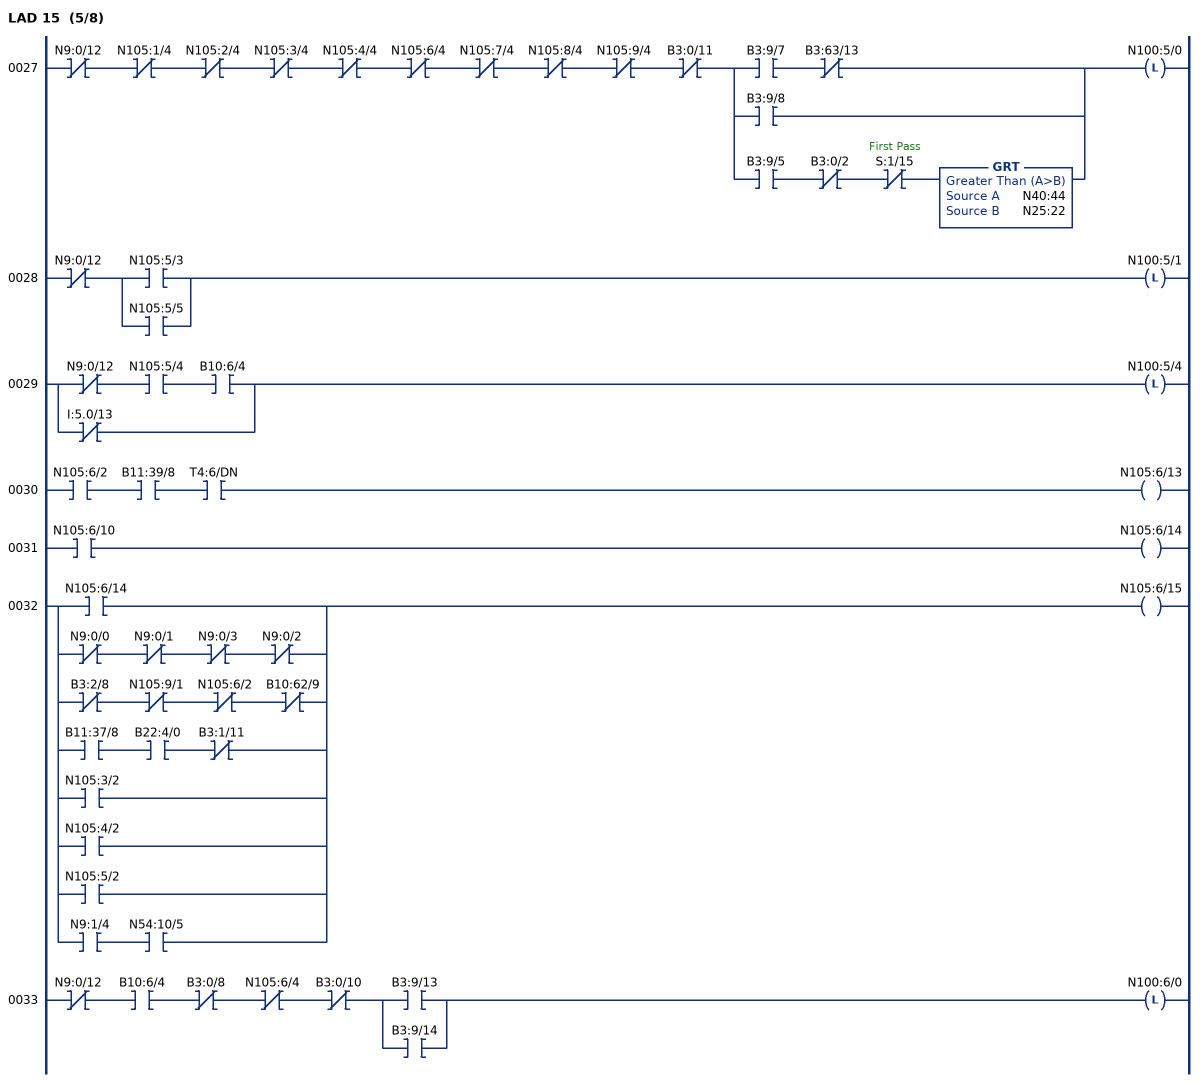
% Rung: 27 %
SOR XIO N9:0/12 XIO N105:1/4 XIO N105:2/4 XIO N105:3/4 XIO N105:4/4 XIO N105:6/4 XIO N105:7/4 XIO N105:8/4 XIO N105:9/4 XIO B3:0/11 BST XIC B3:9/7 XIO B3:63/13 NXB XIC B3:9/8 NXB XIC B3:9/5 XIO B3:0/2 XIO S:1/15 GRT N40:44 N25:22 BND OTL N100:5/0 EOR
%   S:1/15  "First Pass" %
% Rung: 28 %
SOR XIO N9:0/12 BST XIC N105:5/3 NXB XIC N105:5/5 BND OTL N100:5/1 EOR
% Rung: 29 %
SOR BST XIO N9:0/12 XIC N105:5/4 XIC B10:6/4 NXB XIO I:5.0/13 BND OTL N100:5/4 EOR
% Rung: 30 %
SOR XIC N105:6/2 XIC B11:39/8 XIC T4:6/DN OTE N105:6/13 EOR
% Rung: 31 %
SOR XIC N105:6/10 OTE N105:6/14 EOR
% Rung: 32 %
SOR BST XIC N105:6/14 NXB XIO N9:0/0 XIO N9:0/1 XIO N9:0/3 XIO N9:0/2 NXB XIO B3:2/8 XIO N105:9/1 XIO N105:6/2 XIO B10:62/9 NXB XIC B11:37/8 XIC B22:4/0 XIO B3:1/11 NXB XIC N105:3/2 NXB XIC N105:4/2 NXB XIC N105:5/2 NXB XIC N9:1/4 XIC N54:10/5 BND OTE N105:6/15 EOR
% Rung: 33 %
SOR XIO N9:0/12 XIC B10:6/4 XIO B3:0/8 XIO N105:6/4 XIO B3:0/10 BST XIC B3:9/13 NXB XIC B3:9/14 BND OTL N100:6/0 EOR

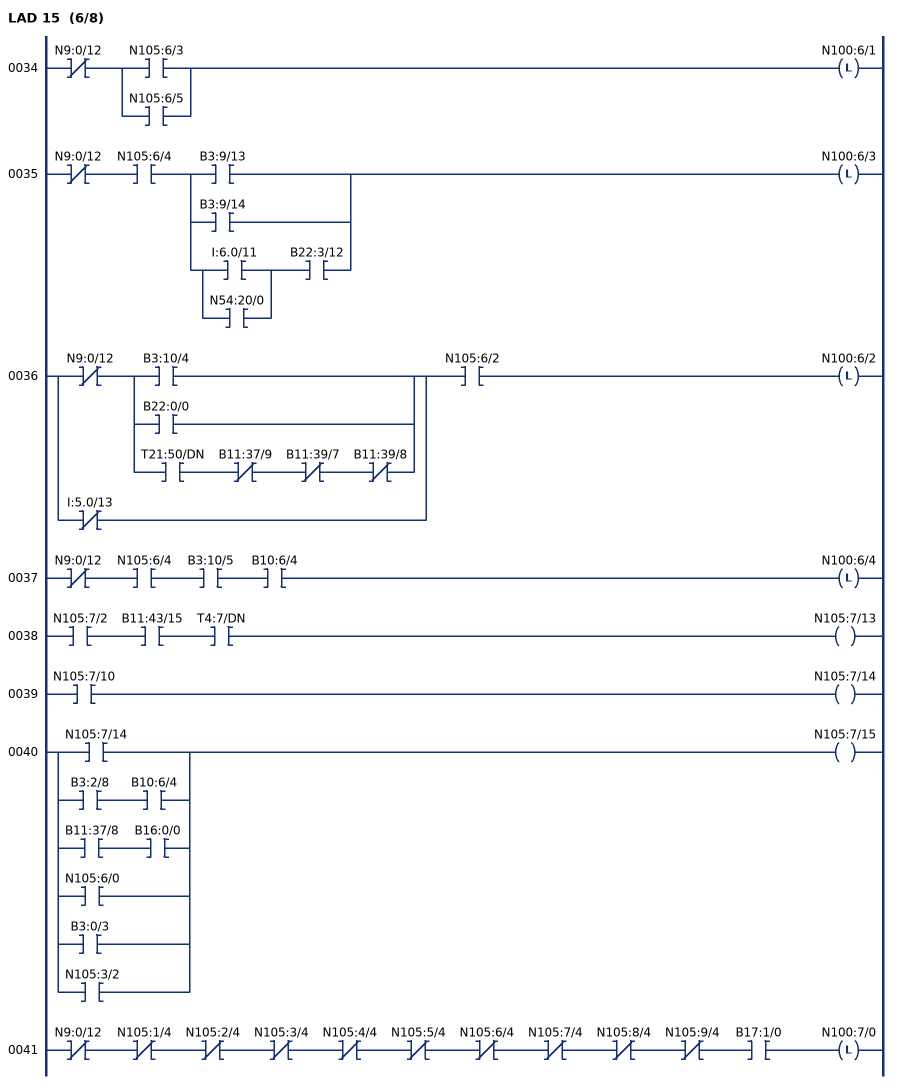
% Rung: 34 %
SOR XIO N9:0/12 BST XIC N105:6/3 NXB XIC N105:6/5 BND OTL N100:6/1 EOR
% Rung: 35 %
SOR XIO N9:0/12 XIC N105:6/4 BST XIC B3:9/13 NXB XIC B3:9/14 NXB BST XIC I:6.0/11 NXB XIC N54:20/0 BND XIC B22:3/12 BND OTL N100:6/3 EOR
% Rung: 36 %
SOR BST XIO N9:0/12 BST XIC B3:10/4 NXB XIC B22:0/0 NXB XIC T21:50/DN XIO B11:37/9 XIO B11:39/7 XIO B11:39/8 BND NXB XIO I:5.0/13 BND XIC N105:6/2 OTL N100:6/2 EOR
% Rung: 37 %
SOR XIO N9:0/12 XIC N105:6/4 XIC B3:10/5 XIC B10:6/4 OTL N100:6/4 EOR
% Rung: 38 %
SOR XIC N105:7/2 XIC B11:43/15 XIC T4:7/DN OTE N105:7/13 EOR
% Rung: 39 %
SOR XIC N105:7/10 OTE N105:7/14 EOR
% Rung: 40 %
SOR BST XIC N105:7/14 NXB XIC B3:2/8 XIC B10:6/4 NXB XIC B11:37/8 XIC B16:0/0 NXB XIC N105:6/0 NXB XIC B3:0/3 NXB XIC N105:3/2 BND OTE N105:7/15 EOR
% Rung: 41 %
SOR XIO N9:0/12 XIO N105:1/4 XIO N105:2/4 XIO N105:3/4 XIO N105:4/4 XIO N105:5/4 XIO N105:6/4 XIO N105:7/4 XIO N105:8/4 XIO N105:9/4 XIC B17:1/0 OTL N100:7/0 EOR

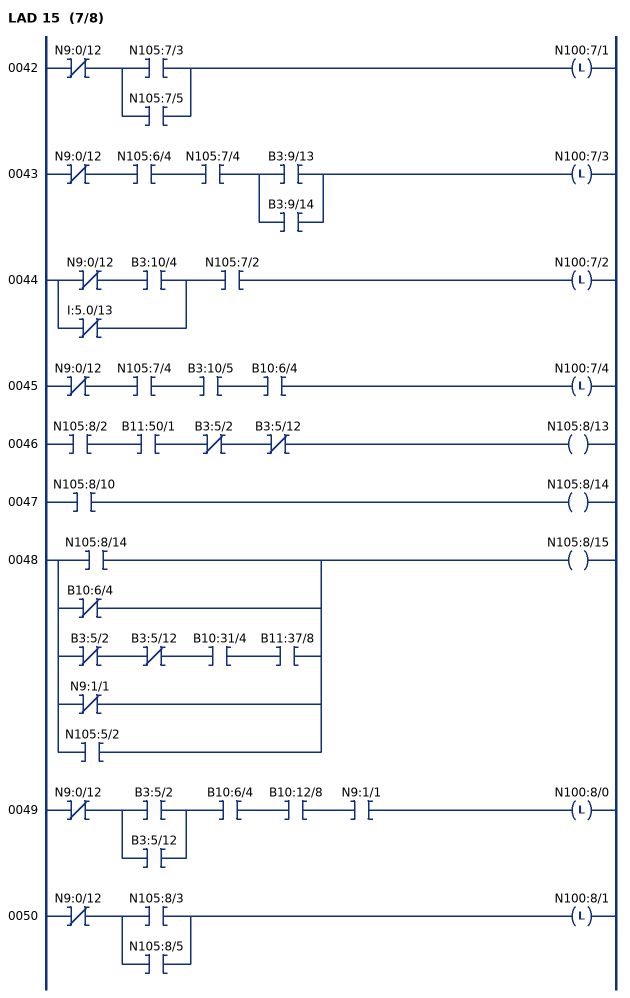
% Rung: 42 %
SOR XIO N9:0/12 BST XIC N105:7/3 NXB XIC N105:7/5 BND OTL N100:7/1 EOR
% Rung: 43 %
SOR XIO N9:0/12 XIC N105:6/4 XIC N105:7/4 BST XIC B3:9/13 NXB XIC B3:9/14 BND OTL N100:7/3 EOR
% Rung: 44 %
SOR BST XIO N9:0/12 XIC B3:10/4 NXB XIO I:5.0/13 BND XIC N105:7/2 OTL N100:7/2 EOR
% Rung: 45 %
SOR XIO N9:0/12 XIC N105:7/4 XIC B3:10/5 XIC B10:6/4 OTL N100:7/4 EOR
% Rung: 46 %
SOR XIC N105:8/2 XIC B11:50/1 XIO B3:5/2 XIO B3:5/12 OTE N105:8/13 EOR
% Rung: 47 %
SOR XIC N105:8/10 OTE N105:8/14 EOR
% Rung: 48 %
SOR BST XIC N105:8/14 NXB XIO B10:6/4 NXB XIO B3:5/2 XIO B3:5/12 XIC B10:31/4 XIC B11:37/8 NXB XIO N9:1/1 NXB XIC N105:5/2 BND OTE N105:8/15 EOR
% Rung: 49 %
SOR XIO N9:0/12 BST XIC B3:5/2 NXB XIC B3:5/12 BND XIC B10:6/4 XIC B10:12/8 XIC N9:1/1 OTL N100:8/0 EOR
% Rung: 50 %
SOR XIO N9:0/12 BST XIC N105:8/3 NXB XIC N105:8/5 BND OTL N100:8/1 EOR

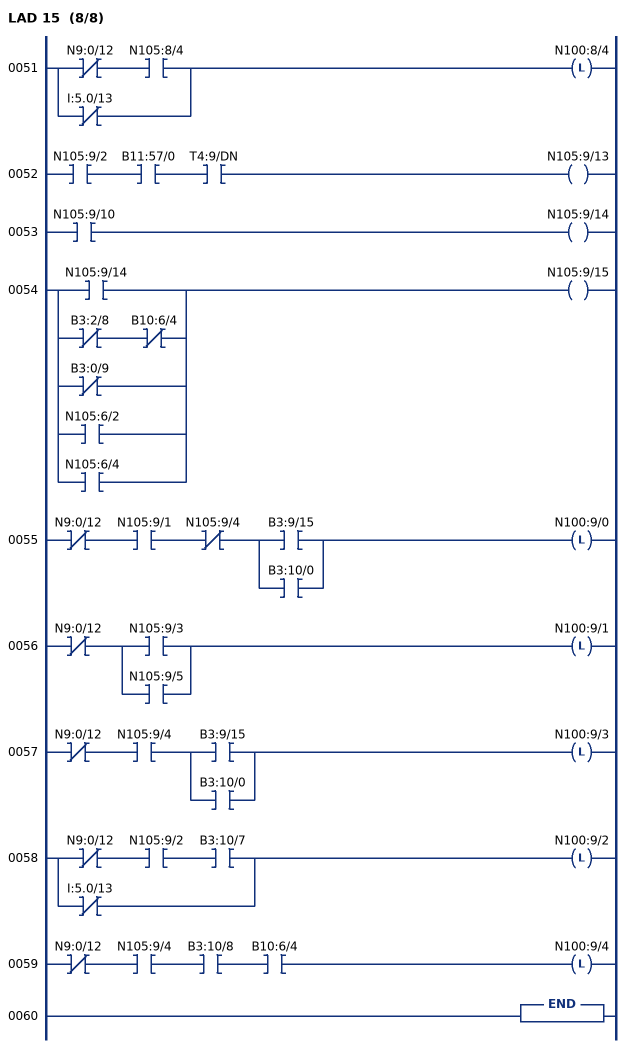
% Rung: 51 %
SOR BST XIO N9:0/12 XIC N105:8/4 NXB XIO I:5.0/13 BND OTL N100:8/4 EOR
% Rung: 52 %
SOR XIC N105:9/2 XIC B11:57/0 XIC T4:9/DN OTE N105:9/13 EOR
% Rung: 53 %
SOR XIC N105:9/10 OTE N105:9/14 EOR
% Rung: 54 %
SOR BST XIC N105:9/14 NXB XIO B3:2/8 XIO B10:6/4 NXB XIO B3:0/9 NXB XIC N105:6/2 NXB XIC N105:6/4 BND OTE N105:9/15 EOR
% Rung: 55 %
SOR XIO N9:0/12 XIC N105:9/1 XIO N105:9/4 BST XIC B3:9/15 NXB XIC B3:10/0 BND OTL N100:9/0 EOR
% Rung: 56 %
SOR XIO N9:0/12 BST XIC N105:9/3 NXB XIC N105:9/5 BND OTL N100:9/1 EOR
% Rung: 57 %
SOR XIO N9:0/12 XIC N105:9/4 BST XIC B3:9/15 NXB XIC B3:10/0 BND OTL N100:9/3 EOR
% Rung: 58 %
SOR BST XIO N9:0/12 XIC N105:9/2 XIC B3:10/7 NXB XIO I:5.0/13 BND OTL N100:9/2 EOR
% Rung: 59 %
SOR XIO N9:0/12 XIC N105:9/4 XIC B3:10/8 XIC B10:6/4 OTL N100:9/4 EOR
% Rung: 60 %
SOR END EOR

LADDER 16
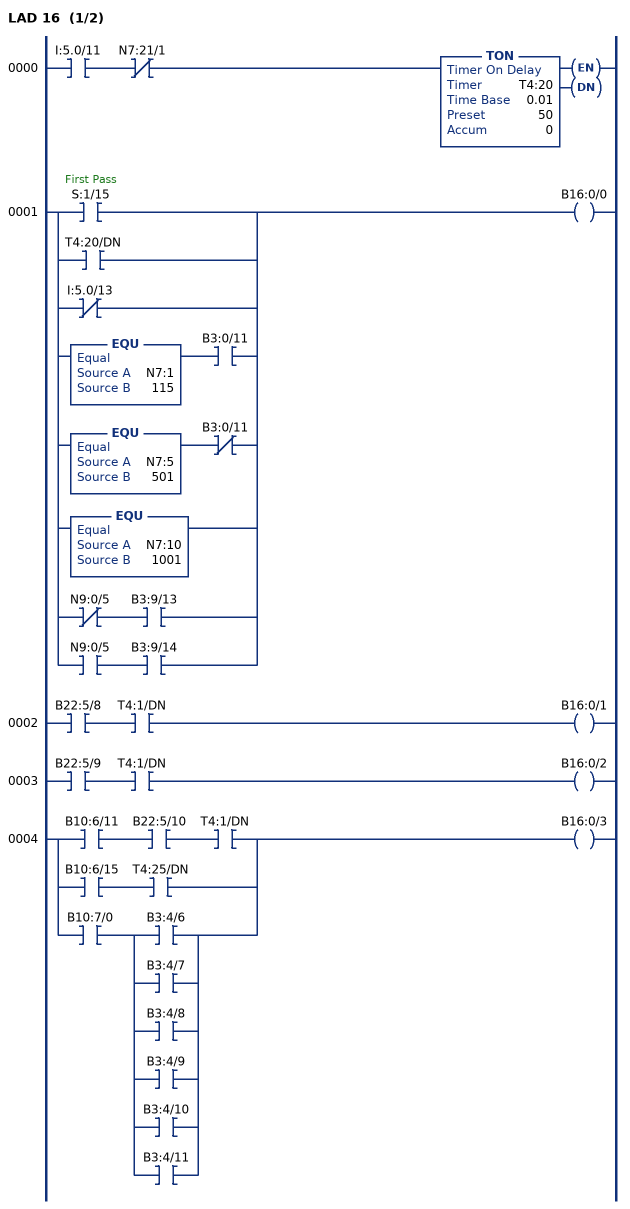
% Rung: 0 %
SOR XIC I:5.0/11 XIO N7:21/1 TON T4:20 0.01 50 0 EOR
% Rung: 1 %
SOR BST BST XIC S:1/15 NXB XIC T4:20/DN BND NXB XIO I:5.0/13 NXB EQU N7:1 115 XIC B3:0/11 NXB EQU N7:5 501 XIO B3:0/11 NXB EQU N7:10 1001 NXB XIO N9:0/5 XIC B3:9/13 NXB XIC N9:0/5 XIC B3:9/14 BND OTE B16:0/0 EOR
%   S:1/15  "First Pass" %
% Rung: 2 %
SOR XIC B22:5/8 XIC T4:1/DN OTE B16:0/1 EOR
% Rung: 3 %
SOR XIC B22:5/9 XIC T4:1/DN OTE B16:0/2 EOR
% Rung: 4 %
SOR BST XIC B10:6/11 XIC B22:5/10 XIC T4:1/DN NXB XIC B10:6/15 XIC T4:25/DN NXB XIC B10:7/0 BST XIC B3:4/6 NXB XIC B3:4/7 NXB XIC B3:4/8 NXB XIC B3:4/9 NXB XIC B3:4/10 NXB XIC B3:4/11 BND BND OTE B16:0/3 EOR

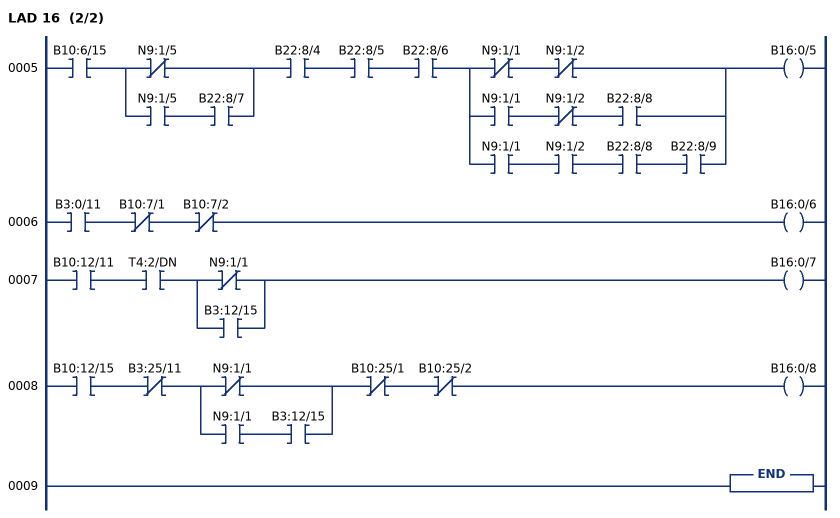
% Rung: 5 %
SOR XIC B10:6/15 BST XIO N9:1/5 NXB XIC N9:1/5 XIC B22:8/7 BND XIC B22:8/4 XIC B22:8/5 XIC B22:8/6 BST XIO N9:1/1 XIO N9:1/2 NXB XIC N9:1/1 XIO N9:1/2 XIC B22:8/8 NXB XIC N9:1/1 XIC N9:1/2 XIC B22:8/8 XIC B22:8/9 BND OTE B16:0/5 EOR
% Rung: 6 %
SOR XIC B3:0/11 XIO B10:7/1 XIO B10:7/2 OTE B16:0/6 EOR
% Rung: 7 %
SOR XIC B10:12/11 XIC T4:2/DN BST XIO N9:1/1 NXB XIC B3:12/15 BND OTE B16:0/7 EOR
% Rung: 8 %
SOR XIC B10:12/15 XIO B3:25/11 BST XIO N9:1/1 NXB XIC N9:1/1 XIC B3:12/15 BND XIO B10:25/1 XIO B10:25/2 OTE B16:0/8 EOR
% Rung: 9 %
SOR END EOR

LADDER 17
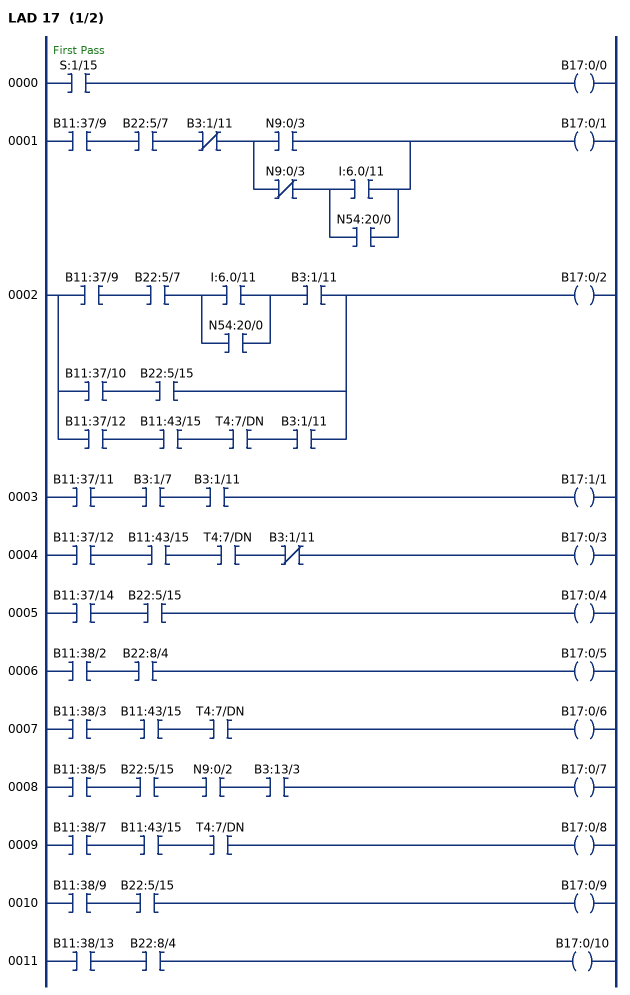
% Rung: 0 %
SOR XIC S:1/15 OTE B17:0/0 EOR
%   S:1/15  "First Pass" %
% Rung: 1 %
SOR XIC B11:37/9 XIC B22:5/7 XIO B3:1/11 BST XIC N9:0/3 NXB XIO N9:0/3 BST XIC I:6.0/11 NXB XIC N54:20/0 BND BND OTE B17:0/1 EOR
% Rung: 2 %
SOR BST XIC B11:37/9 XIC B22:5/7 BST XIC I:6.0/11 NXB XIC N54:20/0 BND XIC B3:1/11 NXB XIC B11:37/10 XIC B22:5/15 NXB XIC B11:37/12 XIC B11:43/15 XIC T4:7/DN XIC B3:1/11 BND OTE B17:0/2 EOR
% Rung: 3 %
SOR XIC B11:37/11 XIC B3:1/7 XIC B3:1/11 OTE B17:1/1 EOR
% Rung: 4 %
SOR XIC B11:37/12 XIC B11:43/15 XIC T4:7/DN XIO B3:1/11 OTE B17:0/3 EOR
% Rung: 5 %
SOR XIC B11:37/14 XIC B22:5/15 OTE B17:0/4 EOR
% Rung: 6 %
SOR XIC B11:38/2 XIC B22:8/4 OTE B17:0/5 EOR
% Rung: 7 %
SOR XIC B11:38/3 XIC B11:43/15 XIC T4:7/DN OTE B17:0/6 EOR
% Rung: 8 %
SOR XIC B11:38/5 XIC B22:5/15 XIC N9:0/2 XIC B3:13/3 OTE B17:0/7 EOR
% Rung: 9 %
SOR XIC B11:38/7 XIC B11:43/15 XIC T4:7/DN OTE B17:0/8 EOR
% Rung: 10 %
SOR XIC B11:38/9 XIC B22:5/15 OTE B17:0/9 EOR
% Rung: 11 %
SOR XIC B11:38/13 XIC B22:8/4 OTE B17:0/10 EOR

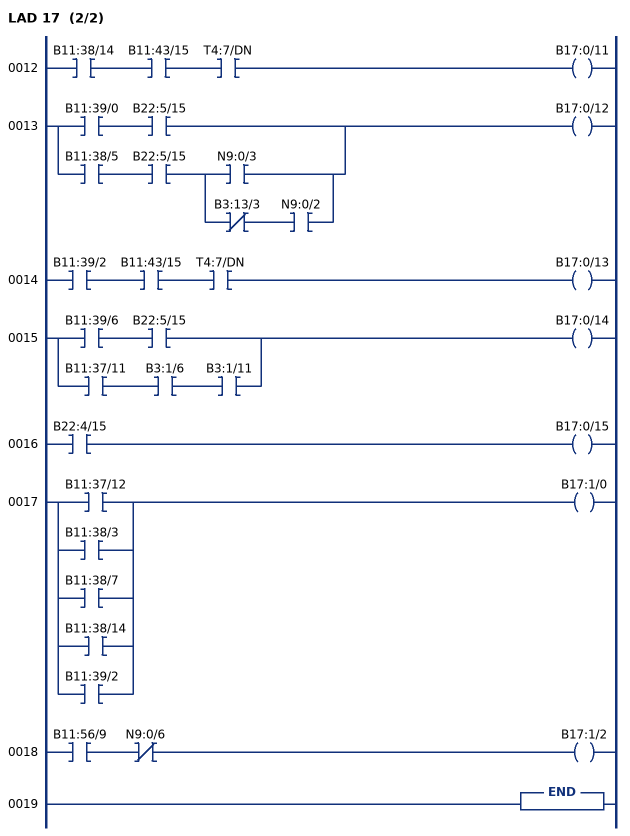
% Rung: 12 %
SOR XIC B11:38/14 XIC B11:43/15 XIC T4:7/DN OTE B17:0/11 EOR
% Rung: 13 %
SOR BST XIC B11:39/0 XIC B22:5/15 NXB XIC B11:38/5 XIC B22:5/15 BST XIC N9:0/3 NXB XIO B3:13/3 XIC N9:0/2 BND BND OTE B17:0/12 EOR
% Rung: 14 %
SOR XIC B11:39/2 XIC B11:43/15 XIC T4:7/DN OTE B17:0/13 EOR
% Rung: 15 %
SOR BST XIC B11:39/6 XIC B22:5/15 NXB XIC B11:37/11 XIC B3:1/6 XIC B3:1/11 BND OTE B17:0/14 EOR
% Rung: 16 %
SOR XIC B22:4/15 OTE B17:0/15 EOR
% Rung: 17 %
SOR BST XIC B11:37/12 NXB XIC B11:38/3 NXB XIC B11:38/7 NXB XIC B11:38/14 NXB XIC B11:39/2 BND OTE B17:1/0 EOR
% Rung: 18 %
SOR XIC B11:56/9 XIO N9:0/6 OTE B17:1/2 EOR
% Rung: 19 %
SOR END EOR

LADDER 21
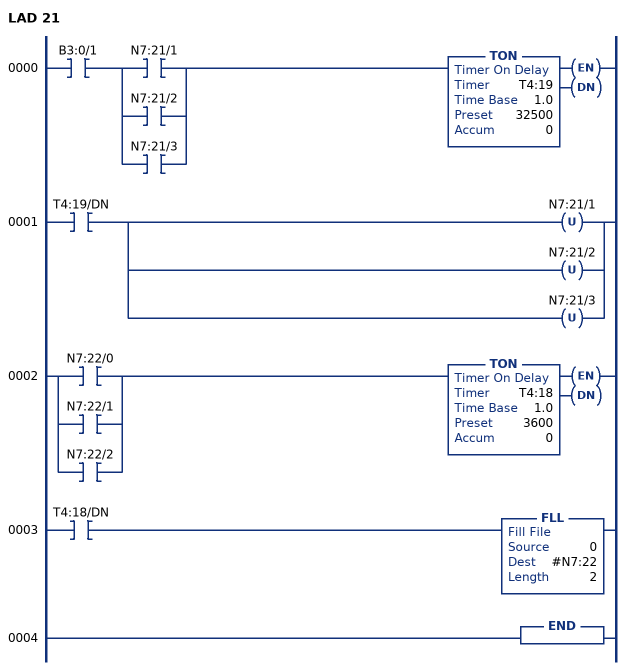
% Rung: 0 %
SOR XIC B3:0/1 BST XIC N7:21/1 NXB XIC N7:21/2 NXB XIC N7:21/3 BND TON T4:19 1.0 32500 0 EOR
% Rung: 1 %
SOR XIC T4:19/DN BST OTU N7:21/1 NXB OTU N7:21/2 NXB OTU N7:21/3 BND EOR
% Rung: 2 %
SOR BST XIC N7:22/0 NXB XIC N7:22/1 NXB XIC N7:22/2 BND TON T4:18 1.0 3600 0 EOR
% Rung: 3 %
SOR XIC T4:18/DN FLL 0 #N7:22 2 EOR
% Rung: 4 %
SOR END EOR

LADDER 22
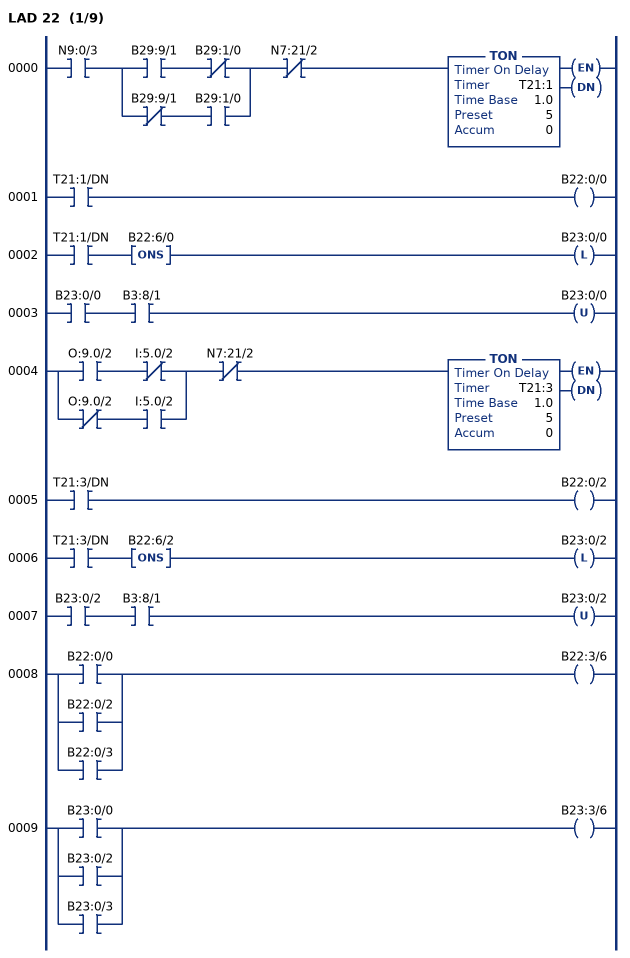
% Rung: 0 %
SOR XIC N9:0/3 BST XIC B29:9/1 XIO B29:1/0 NXB XIO B29:9/1 XIC B29:1/0 BND XIO N7:21/2 TON T21:1 1.0 5 0 EOR
% Rung: 1 %
SOR XIC T21:1/DN OTE B22:0/0 EOR
% Rung: 2 %
SOR XIC T21:1/DN OSR B22:6/0 OTL B23:0/0 EOR
% Rung: 3 %
SOR XIC B23:0/0 XIC B3:8/1 OTU B23:0/0 EOR
% Rung: 4 %
SOR BST XIC O:9.0/2 XIO I:5.0/2 NXB XIO O:9.0/2 XIC I:5.0/2 BND XIO N7:21/2 TON T21:3 1.0 5 0 EOR
% Rung: 5 %
SOR XIC T21:3/DN OTE B22:0/2 EOR
% Rung: 6 %
SOR XIC T21:3/DN OSR B22:6/2 OTL B23:0/2 EOR
% Rung: 7 %
SOR XIC B23:0/2 XIC B3:8/1 OTU B23:0/2 EOR
% Rung: 8 %
SOR BST XIC B22:0/0 NXB XIC B22:0/2 NXB XIC B22:0/3 BND OTE B22:3/6 EOR
% Rung: 9 %
SOR BST XIC B23:0/0 NXB XIC B23:0/2 NXB XIC B23:0/3 BND OTE B23:3/6 EOR

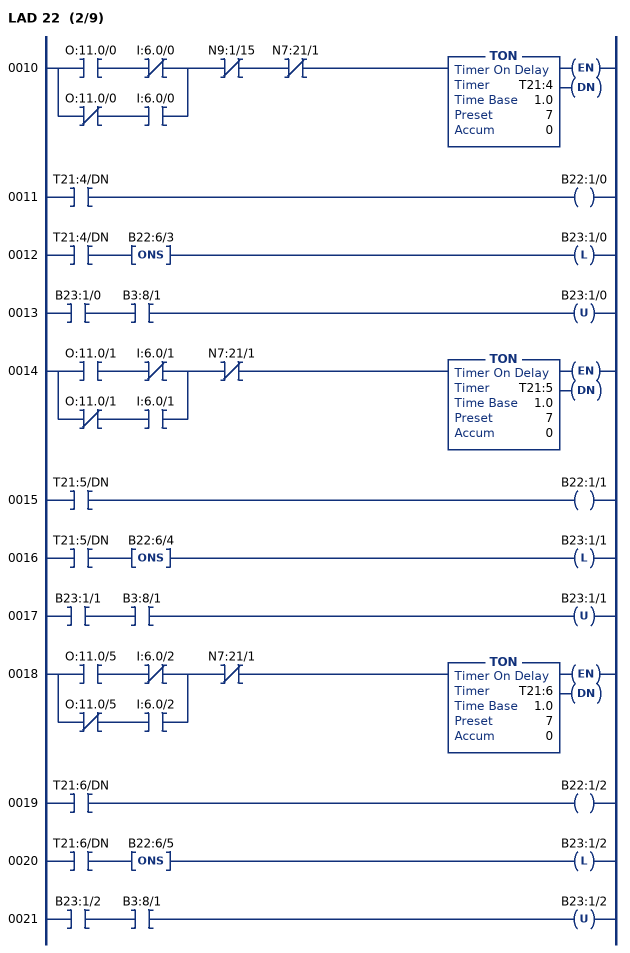
% Rung: 10 %
SOR BST XIC O:11.0/0 XIO I:6.0/0 NXB XIO O:11.0/0 XIC I:6.0/0 BND XIO N9:1/15 XIO N7:21/1 TON T21:4 1.0 7 0 EOR
% Rung: 11 %
SOR XIC T21:4/DN OTE B22:1/0 EOR
% Rung: 12 %
SOR XIC T21:4/DN OSR B22:6/3 OTL B23:1/0 EOR
% Rung: 13 %
SOR XIC B23:1/0 XIC B3:8/1 OTU B23:1/0 EOR
% Rung: 14 %
SOR BST XIC O:11.0/1 XIO I:6.0/1 NXB XIO O:11.0/1 XIC I:6.0/1 BND XIO N7:21/1 TON T21:5 1.0 7 0 EOR
% Rung: 15 %
SOR XIC T21:5/DN OTE B22:1/1 EOR
% Rung: 16 %
SOR XIC T21:5/DN OSR B22:6/4 OTL B23:1/1 EOR
% Rung: 17 %
SOR XIC B23:1/1 XIC B3:8/1 OTU B23:1/1 EOR
% Rung: 18 %
SOR BST XIC O:11.0/5 XIO I:6.0/2 NXB XIO O:11.0/5 XIC I:6.0/2 BND XIO N7:21/1 TON T21:6 1.0 7 0 EOR
% Rung: 19 %
SOR XIC T21:6/DN OTE B22:1/2 EOR
% Rung: 20 %
SOR XIC T21:6/DN OSR B22:6/5 OTL B23:1/2 EOR
% Rung: 21 %
SOR XIC B23:1/2 XIC B3:8/1 OTU B23:1/2 EOR

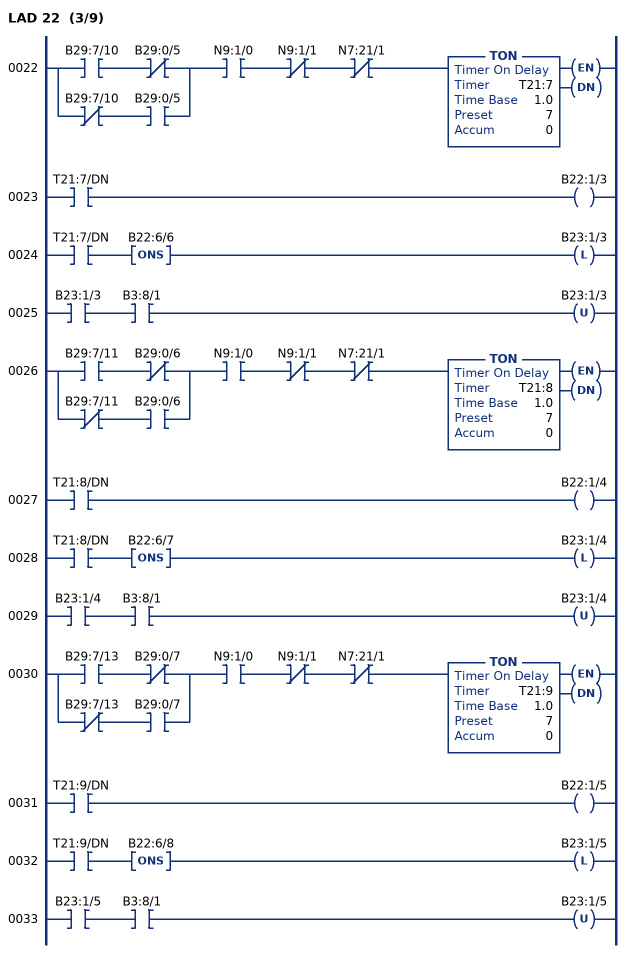
% Rung: 22 %
SOR BST XIC B29:7/10 XIO B29:0/5 NXB XIO B29:7/10 XIC B29:0/5 BND XIC N9:1/0 XIO N9:1/1 XIO N7:21/1 TON T21:7 1.0 7 0 EOR
% Rung: 23 %
SOR XIC T21:7/DN OTE B22:1/3 EOR
% Rung: 24 %
SOR XIC T21:7/DN OSR B22:6/6 OTL B23:1/3 EOR
% Rung: 25 %
SOR XIC B23:1/3 XIC B3:8/1 OTU B23:1/3 EOR
% Rung: 26 %
SOR BST XIC B29:7/11 XIO B29:0/6 NXB XIO B29:7/11 XIC B29:0/6 BND XIC N9:1/0 XIO N9:1/1 XIO N7:21/1 TON T21:8 1.0 7 0 EOR
% Rung: 27 %
SOR XIC T21:8/DN OTE B22:1/4 EOR
% Rung: 28 %
SOR XIC T21:8/DN OSR B22:6/7 OTL B23:1/4 EOR
% Rung: 29 %
SOR XIC B23:1/4 XIC B3:8/1 OTU B23:1/4 EOR
% Rung: 30 %
SOR BST XIC B29:7/13 XIO B29:0/7 NXB XIO B29:7/13 XIC B29:0/7 BND XIC N9:1/0 XIO N9:1/1 XIO N7:21/1 TON T21:9 1.0 7 0 EOR
% Rung: 31 %
SOR XIC T21:9/DN OTE B22:1/5 EOR
% Rung: 32 %
SOR XIC T21:9/DN OSR B22:6/8 OTL B23:1/5 EOR
% Rung: 33 %
SOR XIC B23:1/5 XIC B3:8/1 OTU B23:1/5 EOR

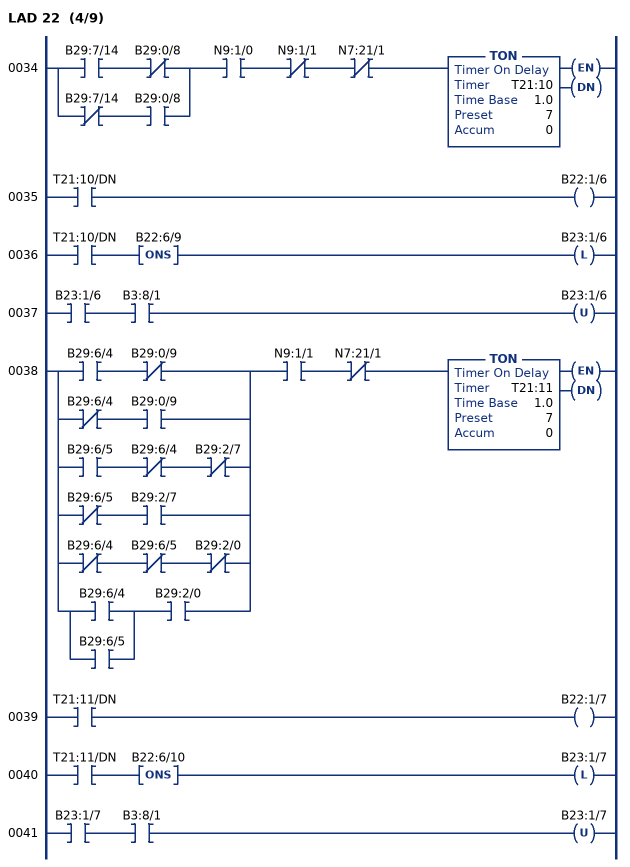
% Rung: 34 %
SOR BST XIC B29:7/14 XIO B29:0/8 NXB XIO B29:7/14 XIC B29:0/8 BND XIC N9:1/0 XIO N9:1/1 XIO N7:21/1 TON T21:10 1.0 7 0 EOR
% Rung: 35 %
SOR XIC T21:10/DN OTE B22:1/6 EOR
% Rung: 36 %
SOR XIC T21:10/DN OSR B22:6/9 OTL B23:1/6 EOR
% Rung: 37 %
SOR XIC B23:1/6 XIC B3:8/1 OTU B23:1/6 EOR
% Rung: 38 %
SOR BST XIC B29:6/4 XIO B29:0/9 NXB XIO B29:6/4 XIC B29:0/9 NXB XIC B29:6/5 XIO B29:6/4 XIO B29:2/7 NXB XIO B29:6/5 XIC B29:2/7 NXB XIO B29:6/4 XIO B29:6/5 XIO B29:2/0 NXB BST XIC B29:6/4 NXB XIC B29:6/5 BND XIC B29:2/0 BND XIC N9:1/1 XIO N7:21/1 TON T21:11 1.0 7 0 EOR
% Rung: 39 %
SOR XIC T21:11/DN OTE B22:1/7 EOR
% Rung: 40 %
SOR XIC T21:11/DN OSR B22:6/10 OTL B23:1/7 EOR
% Rung: 41 %
SOR XIC B23:1/7 XIC B3:8/1 OTU B23:1/7 EOR

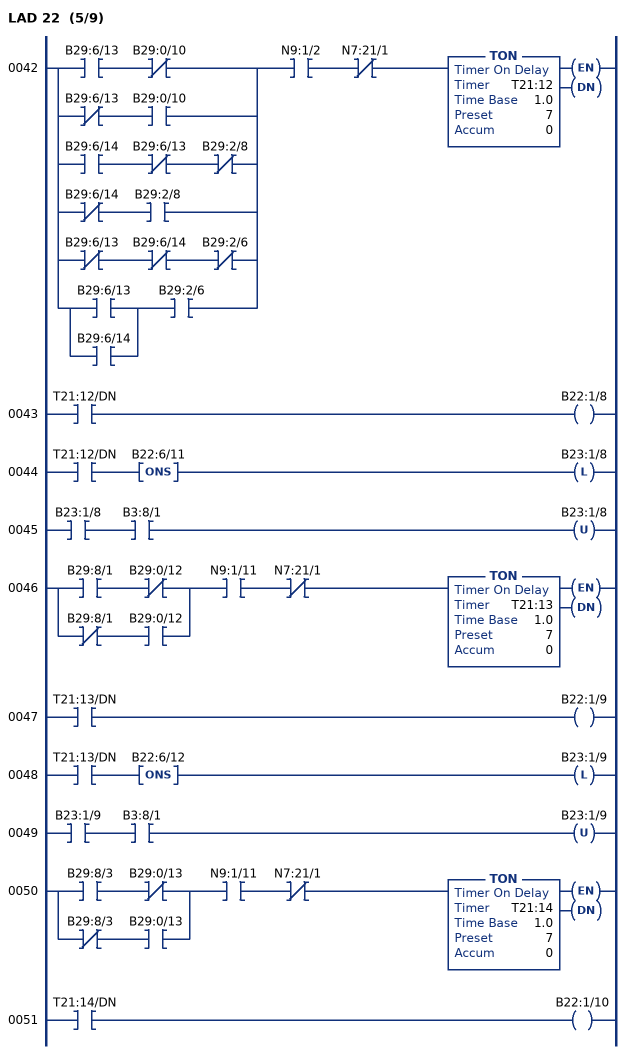
% Rung: 42 %
SOR BST XIC B29:6/13 XIO B29:0/10 NXB XIO B29:6/13 XIC B29:0/10 NXB XIC B29:6/14 XIO B29:6/13 XIO B29:2/8 NXB XIO B29:6/14 XIC B29:2/8 NXB XIO B29:6/13 XIO B29:6/14 XIO B29:2/6 NXB BST XIC B29:6/13 NXB XIC B29:6/14 BND XIC B29:2/6 BND XIC N9:1/2 XIO N7:21/1 TON T21:12 1.0 7 0 EOR
% Rung: 43 %
SOR XIC T21:12/DN OTE B22:1/8 EOR
% Rung: 44 %
SOR XIC T21:12/DN OSR B22:6/11 OTL B23:1/8 EOR
% Rung: 45 %
SOR XIC B23:1/8 XIC B3:8/1 OTU B23:1/8 EOR
% Rung: 46 %
SOR BST XIC B29:8/1 XIO B29:0/12 NXB XIO B29:8/1 XIC B29:0/12 BND XIC N9:1/11 XIO N7:21/1 TON T21:13 1.0 7 0 EOR
% Rung: 47 %
SOR XIC T21:13/DN OTE B22:1/9 EOR
% Rung: 48 %
SOR XIC T21:13/DN OSR B22:6/12 OTL B23:1/9 EOR
% Rung: 49 %
SOR XIC B23:1/9 XIC B3:8/1 OTU B23:1/9 EOR
% Rung: 50 %
SOR BST XIC B29:8/3 XIO B29:0/13 NXB XIO B29:8/3 XIC B29:0/13 BND XIC N9:1/11 XIO N7:21/1 TON T21:14 1.0 7 0 EOR
% Rung: 51 %
SOR XIC T21:14/DN OTE B22:1/10 EOR

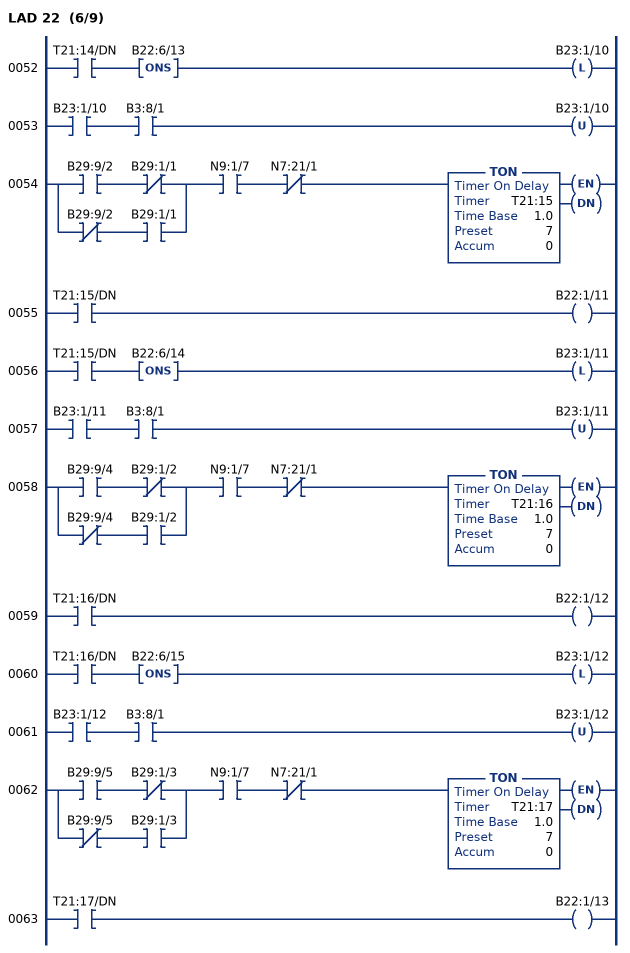
% Rung: 52 %
SOR XIC T21:14/DN OSR B22:6/13 OTL B23:1/10 EOR
% Rung: 53 %
SOR XIC B23:1/10 XIC B3:8/1 OTU B23:1/10 EOR
% Rung: 54 %
SOR BST XIC B29:9/2 XIO B29:1/1 NXB XIO B29:9/2 XIC B29:1/1 BND XIC N9:1/7 XIO N7:21/1 TON T21:15 1.0 7 0 EOR
% Rung: 55 %
SOR XIC T21:15/DN OTE B22:1/11 EOR
% Rung: 56 %
SOR XIC T21:15/DN OSR B22:6/14 OTL B23:1/11 EOR
% Rung: 57 %
SOR XIC B23:1/11 XIC B3:8/1 OTU B23:1/11 EOR
% Rung: 58 %
SOR BST XIC B29:9/4 XIO B29:1/2 NXB XIO B29:9/4 XIC B29:1/2 BND XIC N9:1/7 XIO N7:21/1 TON T21:16 1.0 7 0 EOR
% Rung: 59 %
SOR XIC T21:16/DN OTE B22:1/12 EOR
% Rung: 60 %
SOR XIC T21:16/DN OSR B22:6/15 OTL B23:1/12 EOR
% Rung: 61 %
SOR XIC B23:1/12 XIC B3:8/1 OTU B23:1/12 EOR
% Rung: 62 %
SOR BST XIC B29:9/5 XIO B29:1/3 NXB XIO B29:9/5 XIC B29:1/3 BND XIC N9:1/7 XIO N7:21/1 TON T21:17 1.0 7 0 EOR
% Rung: 63 %
SOR XIC T21:17/DN OTE B22:1/13 EOR

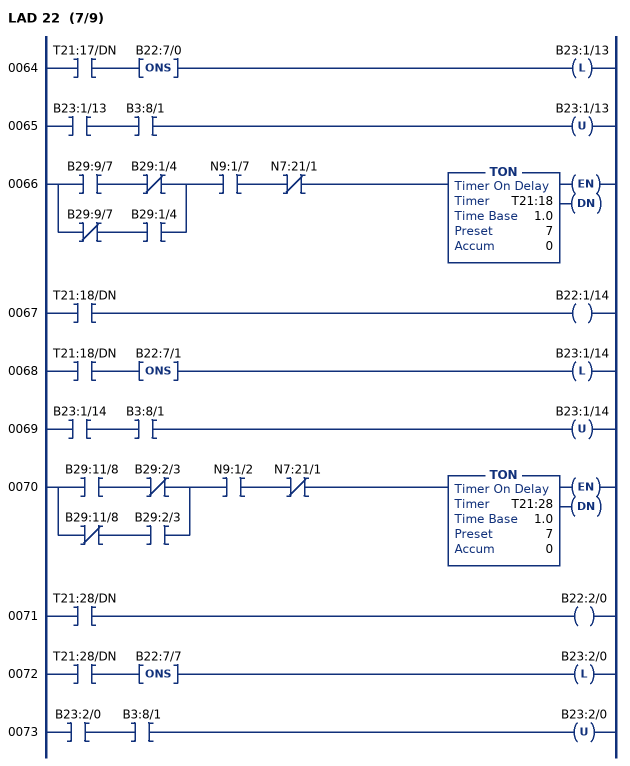
% Rung: 64 %
SOR XIC T21:17/DN OSR B22:7/0 OTL B23:1/13 EOR
% Rung: 65 %
SOR XIC B23:1/13 XIC B3:8/1 OTU B23:1/13 EOR
% Rung: 66 %
SOR BST XIC B29:9/7 XIO B29:1/4 NXB XIO B29:9/7 XIC B29:1/4 BND XIC N9:1/7 XIO N7:21/1 TON T21:18 1.0 7 0 EOR
% Rung: 67 %
SOR XIC T21:18/DN OTE B22:1/14 EOR
% Rung: 68 %
SOR XIC T21:18/DN OSR B22:7/1 OTL B23:1/14 EOR
% Rung: 69 %
SOR XIC B23:1/14 XIC B3:8/1 OTU B23:1/14 EOR
% Rung: 70 %
SOR BST XIC B29:11/8 XIO B29:2/3 NXB XIO B29:11/8 XIC B29:2/3 BND XIC N9:1/2 XIO N7:21/1 TON T21:28 1.0 7 0 EOR
% Rung: 71 %
SOR XIC T21:28/DN OTE B22:2/0 EOR
% Rung: 72 %
SOR XIC T21:28/DN OSR B22:7/7 OTL B23:2/0 EOR
% Rung: 73 %
SOR XIC B23:2/0 XIC B3:8/1 OTU B23:2/0 EOR

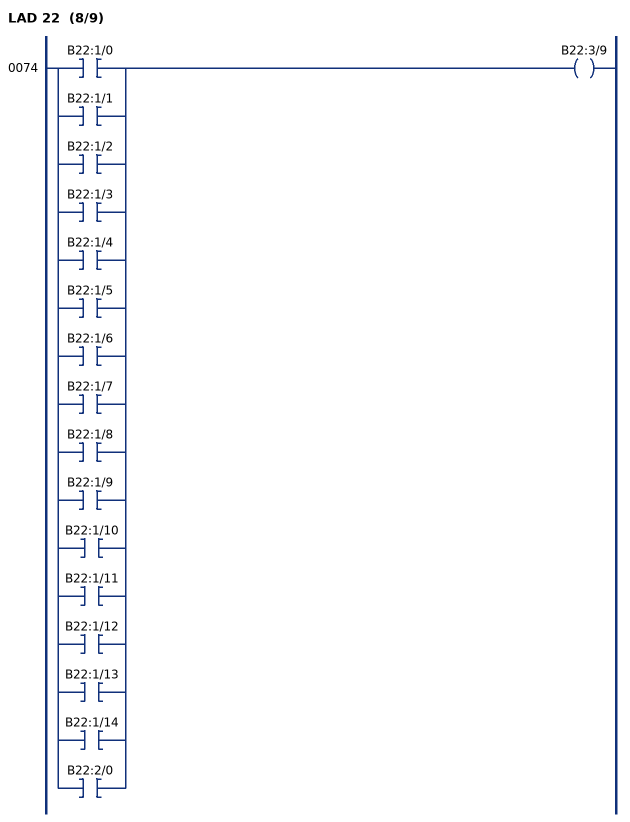
% Rung: 74 %
SOR BST XIC B22:1/0 NXB XIC B22:1/1 NXB XIC B22:1/2 NXB XIC B22:1/3 NXB XIC B22:1/4 NXB XIC B22:1/5 NXB XIC B22:1/6 NXB XIC B22:1/7 NXB XIC B22:1/8 NXB XIC B22:1/9 NXB XIC B22:1/10 NXB XIC B22:1/11 NXB XIC B22:1/12 NXB XIC B22:1/13 NXB XIC B22:1/14 NXB XIC B22:2/0 BND OTE B22:3/9 EOR

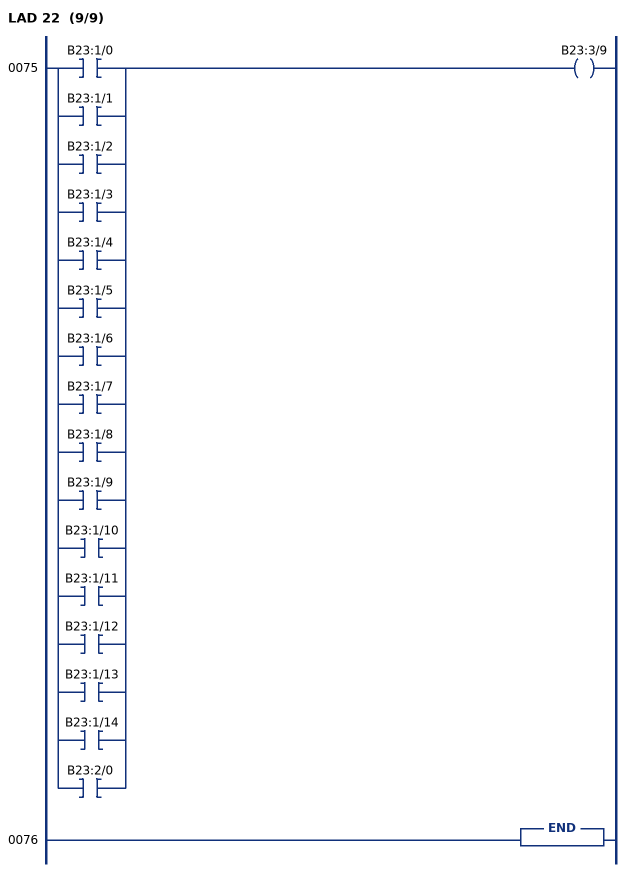
% Rung: 75 %
SOR BST XIC B23:1/0 NXB XIC B23:1/1 NXB XIC B23:1/2 NXB XIC B23:1/3 NXB XIC B23:1/4 NXB XIC B23:1/5 NXB XIC B23:1/6 NXB XIC B23:1/7 NXB XIC B23:1/8 NXB XIC B23:1/9 NXB XIC B23:1/10 NXB XIC B23:1/11 NXB XIC B23:1/12 NXB XIC B23:1/13 NXB XIC B23:1/14 NXB XIC B23:2/0 BND OTE B23:3/9 EOR
% Rung: 76 %
SOR END EOR

LADDER 25
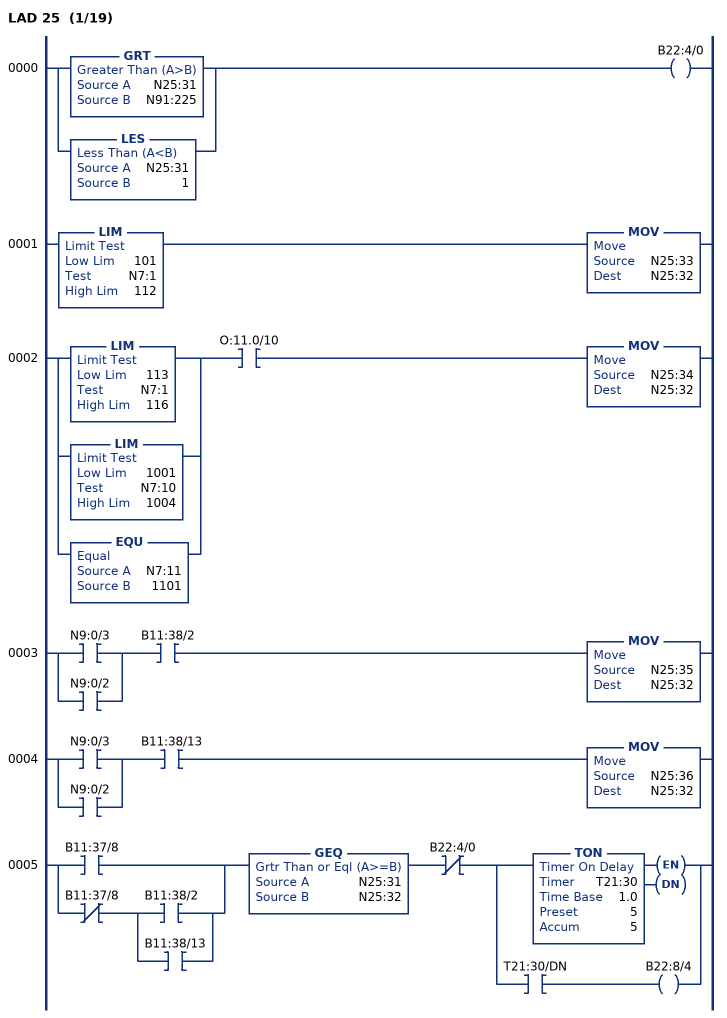
% Rung: 0 %
SOR BST GRT N25:31 N91:225 NXB LES N25:31 1 BND OTE B22:4/0 EOR
% Rung: 1 %
SOR LIM 101 N7:1 112 MOV N25:33 N25:32 EOR
% Rung: 2 %
SOR BST LIM 113 N7:1 116 NXB LIM 1001 N7:10 1004 NXB EQU N7:11 1101 BND XIC O:11.0/10 MOV N25:34 N25:32 EOR
% Rung: 3 %
SOR BST XIC N9:0/3 NXB XIC N9:0/2 BND XIC B11:38/2 MOV N25:35 N25:32 EOR
% Rung: 4 %
SOR BST XIC N9:0/3 NXB XIC N9:0/2 BND XIC B11:38/13 MOV N25:36 N25:32 EOR
% Rung: 5 %
SOR BST XIC B11:37/8 NXB XIO B11:37/8 BST XIC B11:38/2 NXB XIC B11:38/13 BND BND GEQ N25:31 N25:32 XIO B22:4/0 BST TON T21:30 1.0 5 5 NXB XIC T21:30/DN OTE B22:8/4 BND EOR

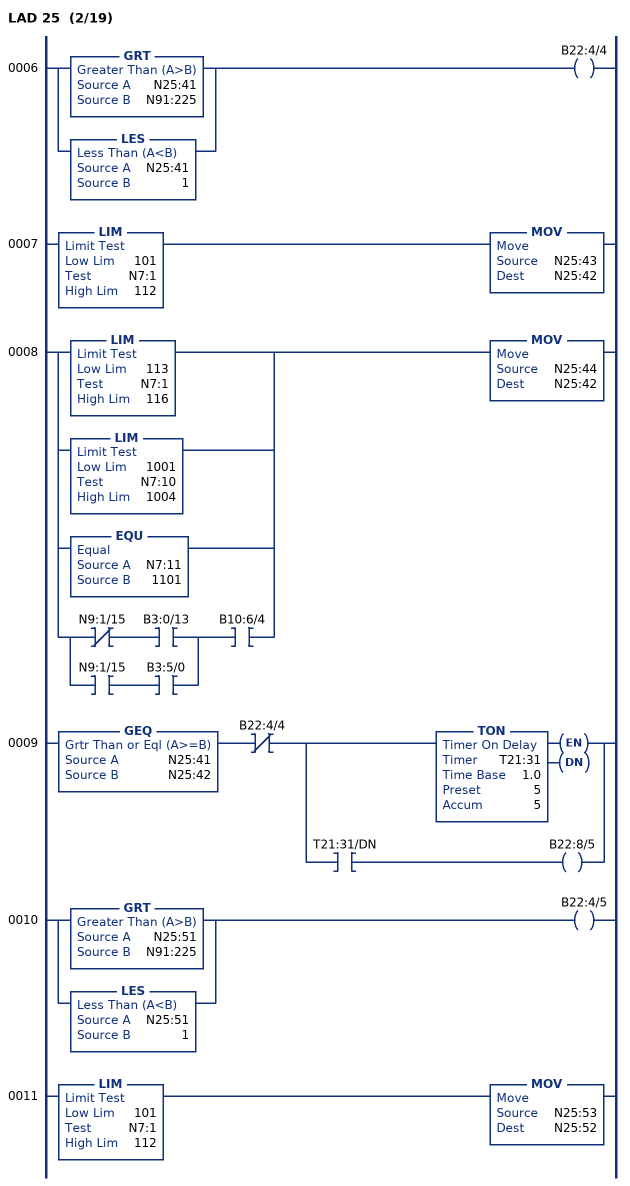
% Rung: 6 %
SOR BST GRT N25:41 N91:225 NXB LES N25:41 1 BND OTE B22:4/4 EOR
% Rung: 7 %
SOR LIM 101 N7:1 112 MOV N25:43 N25:42 EOR
% Rung: 8 %
SOR BST LIM 113 N7:1 116 NXB LIM 1001 N7:10 1004 NXB EQU N7:11 1101 NXB BST XIO N9:1/15 XIC B3:0/13 NXB XIC N9:1/15 XIC B3:5/0 BND XIC B10:6/4 BND MOV N25:44 N25:42 EOR
% Rung: 9 %
SOR GEQ N25:41 N25:42 XIO B22:4/4 BST TON T21:31 1.0 5 5 NXB XIC T21:31/DN OTE B22:8/5 BND EOR
% Rung: 10 %
SOR BST GRT N25:51 N91:225 NXB LES N25:51 1 BND OTE B22:4/5 EOR
% Rung: 11 %
SOR LIM 101 N7:1 112 MOV N25:53 N25:52 EOR

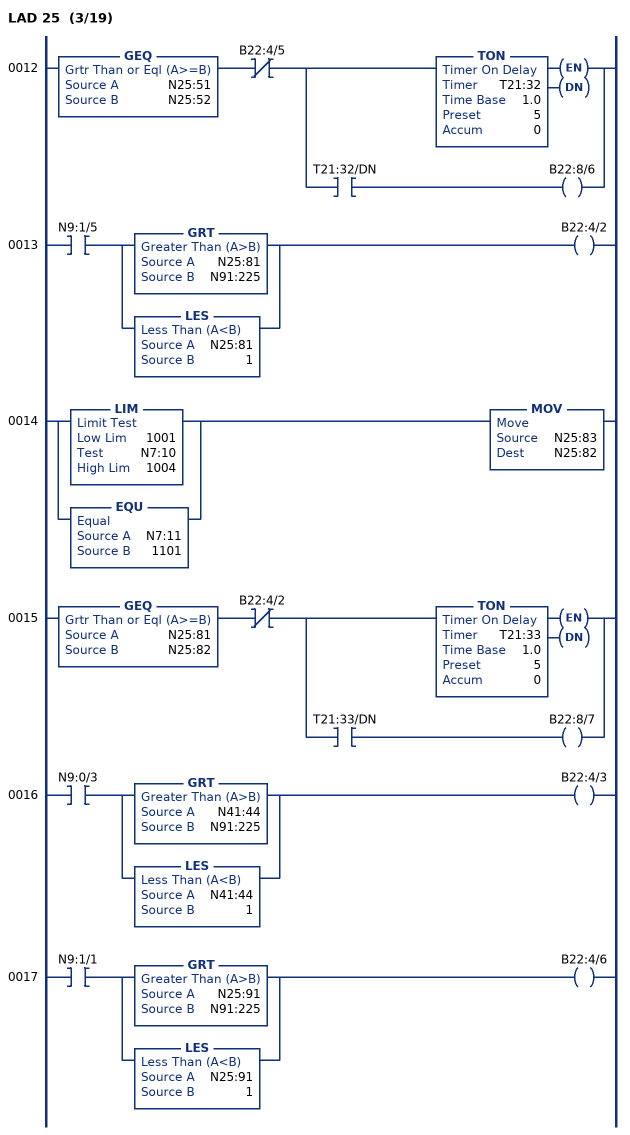
% Rung: 12 %
SOR GEQ N25:51 N25:52 XIO B22:4/5 BST TON T21:32 1.0 5 0 NXB XIC T21:32/DN OTE B22:8/6 BND EOR
% Rung: 13 %
SOR XIC N9:1/5 BST GRT N25:81 N91:225 NXB LES N25:81 1 BND OTE B22:4/2 EOR
% Rung: 14 %
SOR BST LIM 1001 N7:10 1004 NXB EQU N7:11 1101 BND MOV N25:83 N25:82 EOR
% Rung: 15 %
SOR GEQ N25:81 N25:82 XIO B22:4/2 BST TON T21:33 1.0 5 0 NXB XIC T21:33/DN OTE B22:8/7 BND EOR
% Rung: 16 %
SOR XIC N9:0/3 BST GRT N41:44 N91:225 NXB LES N41:44 1 BND OTE B22:4/3 EOR
% Rung: 17 %
SOR XIC N9:1/1 BST GRT N25:91 N91:225 NXB LES N25:91 1 BND OTE B22:4/6 EOR

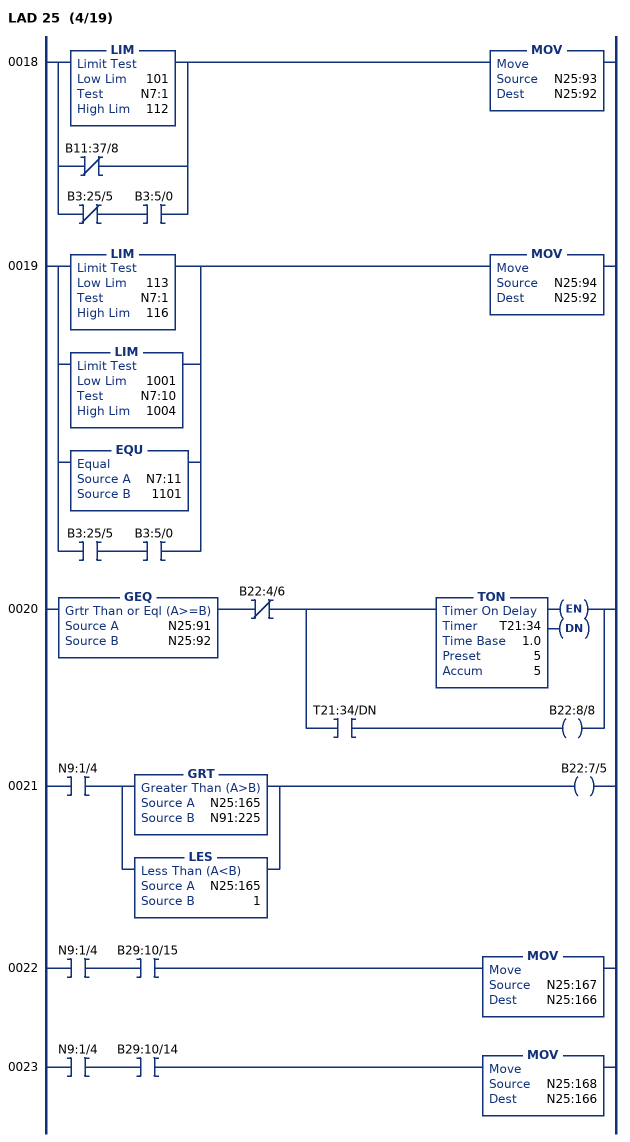
% Rung: 18 %
SOR BST LIM 101 N7:1 112 NXB XIO B11:37/8 NXB XIO B3:25/5 XIC B3:5/0 BND MOV N25:93 N25:92 EOR
% Rung: 19 %
SOR BST LIM 113 N7:1 116 NXB LIM 1001 N7:10 1004 NXB EQU N7:11 1101 NXB XIC B3:25/5 XIC B3:5/0 BND MOV N25:94 N25:92 EOR
% Rung: 20 %
SOR GEQ N25:91 N25:92 XIO B22:4/6 BST TON T21:34 1.0 5 5 NXB XIC T21:34/DN OTE B22:8/8 BND EOR
% Rung: 21 %
SOR XIC N9:1/4 BST GRT N25:165 N91:225 NXB LES N25:165 1 BND OTE B22:7/5 EOR
% Rung: 22 %
SOR XIC N9:1/4 XIC B29:10/15 MOV N25:167 N25:166 EOR
% Rung: 23 %
SOR XIC N9:1/4 XIC B29:10/14 MOV N25:168 N25:166 EOR

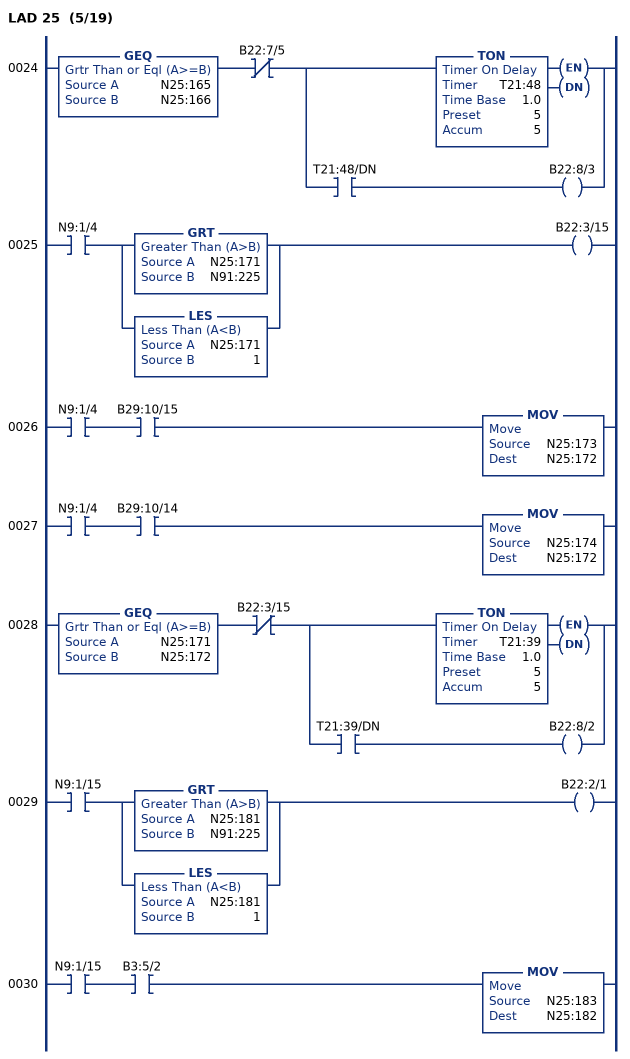
% Rung: 24 %
SOR GEQ N25:165 N25:166 XIO B22:7/5 BST TON T21:48 1.0 5 5 NXB XIC T21:48/DN OTE B22:8/3 BND EOR
% Rung: 25 %
SOR XIC N9:1/4 BST GRT N25:171 N91:225 NXB LES N25:171 1 BND OTE B22:3/15 EOR
% Rung: 26 %
SOR XIC N9:1/4 XIC B29:10/15 MOV N25:173 N25:172 EOR
% Rung: 27 %
SOR XIC N9:1/4 XIC B29:10/14 MOV N25:174 N25:172 EOR
% Rung: 28 %
SOR GEQ N25:171 N25:172 XIO B22:3/15 BST TON T21:39 1.0 5 5 NXB XIC T21:39/DN OTE B22:8/2 BND EOR
% Rung: 29 %
SOR XIC N9:1/15 BST GRT N25:181 N91:225 NXB LES N25:181 1 BND OTE B22:2/1 EOR
% Rung: 30 %
SOR XIC N9:1/15 XIC B3:5/2 MOV N25:183 N25:182 EOR

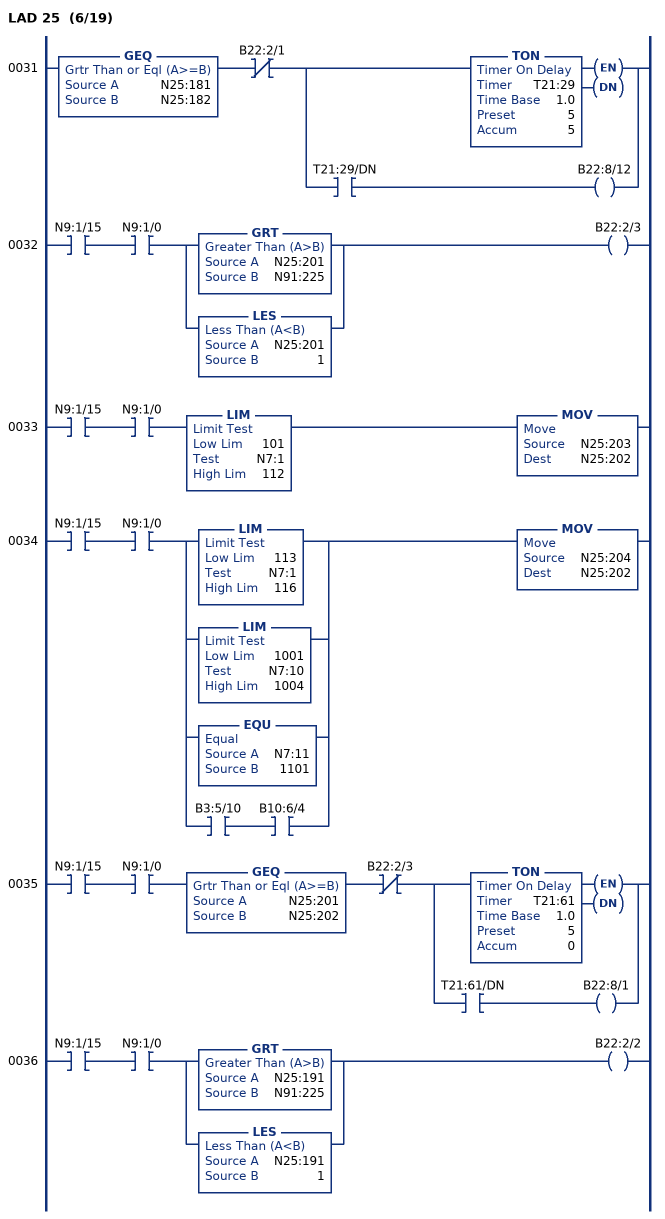
% Rung: 31 %
SOR GEQ N25:181 N25:182 XIO B22:2/1 BST TON T21:29 1.0 5 5 NXB XIC T21:29/DN OTE B22:8/12 BND EOR
% Rung: 32 %
SOR XIC N9:1/15 XIC N9:1/0 BST GRT N25:201 N91:225 NXB LES N25:201 1 BND OTE B22:2/3 EOR
% Rung: 33 %
SOR XIC N9:1/15 XIC N9:1/0 LIM 101 N7:1 112 MOV N25:203 N25:202 EOR
% Rung: 34 %
SOR XIC N9:1/15 XIC N9:1/0 BST LIM 113 N7:1 116 NXB LIM 1001 N7:10 1004 NXB EQU N7:11 1101 NXB XIC B3:5/10 XIC B10:6/4 BND MOV N25:204 N25:202 EOR
% Rung: 35 %
SOR XIC N9:1/15 XIC N9:1/0 GEQ N25:201 N25:202 XIO B22:2/3 BST TON T21:61 1.0 5 0 NXB XIC T21:61/DN OTE B22:8/1 BND EOR
% Rung: 36 %
SOR XIC N9:1/15 XIC N9:1/0 BST GRT N25:191 N91:225 NXB LES N25:191 1 BND OTE B22:2/2 EOR

